// Implicitly generated code : DO NOT EDIT
FUNCTION CheckDivReal : REAL
VAR_INPUT
	divisor:REAL;
END_VAR

// Implicitly generated code : Only an Implementation suggestion
IF divisor = 0 THEN
	CheckDivReal:=1;
	nCheckDivReal := nCheckDivReal + 1;
ELSE
	CheckDivReal:=divisor;
END_IF;

END_FUNCTION

(* stored: Version 1.1.0.1
   POU CheckDivReal: Id {ce0b590d-e089-49e2-b1c9-969f2cbdf1b3}, SpecialFunc CheckDivReal32 *)
